Staubli VAL3: Point2Joint.pgx

public program Point2Joint(pointRx x_pP, jointRx& x_jJDest, bool& x_bRes)
  local point l_pPoint
  local frame l_fFrame
begin



  //如果没有偏移和阵列，直接就进行变换
  if TxtFile:fPofffset.trsf=={0,0,0,0,0,0} and TxtFile:fToffset.trsf=={0,0,0,0,0,0} and TxtFile:fArray.trsf=={0,0,0,0,0,0}

    l_pPoint=x_pP

  else

    link(l_fFrame,world)
    l_fFrame.trsf=TxtFile:fProduct.trsf*TxtFile:fTraj.trsf

    //最原始的点
    l_pPoint.trsf=position(x_pP,world)
    l_pPoint.trsf=!TxtFile:fArray.trsf*!TxtFile:fToffset.trsf*!TxtFile:fTraj.trsf*!TxtFile:fPofffset.trsf*!TxtFile:fProduct.trsf*l_pPoint.trsf
 //   l_pPoint.trsf=
    link(l_pPoint,l_fFrame)
  endIf

  x_bRes=pointToJoint(TxtFile:tCfg,herej(),l_pPoint,x_jJDest)



end
